# EPICS autosave request: eurotherm2k/eurothermModbusLoop_settings.req
$(P)$(Q):D
$(P)$(Q):I
$(P)$(Q):MAN
$(P)$(Q):O
$(P)$(Q):P
$(P)$(Q):PREC
$(P)$(Q):RR
$(P)$(Q):SP
